{attribute 'GeneratedUsingTerminal: EJ2914-0000-0017'}
{attribute addProperty BoxType "EJ2914-0000-0017"}
{attribute addProperty Id "FSoE_InputsFSoE_Inputs_15C2E7B16FSoE_OutputsFSoE_Outputs_C9D9BEFD10"}
{attribute addProperty CRC "556403558"}
{attribute addProperty Size "16"}
TYPE Module_1_FSOE_212A0B66 :
STRUCT
	{attribute addProperty Name "FSoE_Inputs"}
	FSoE_Inputs  : FSoE_Inputs_15C2E7B1;
	{attribute addProperty Name "FSoE_Outputs"}
	FSoE_Outputs  : FSoE_Outputs_C9D9BEFD;
END_STRUCT
END_TYPE

(* stored: Version 1.2.0.0, ProductVersion 3.1.4024.11
   DUT Module_1_FSOE_212A0B66: Id {d6821092-c4d1-4490-aa97-1922803bd70d} *)
